(* IEC 61131-3 sources: Industry-PLC-LLM/data/PLCBEAD_repo/PLCBEAD_PLCEmbed-main/PLC-BEAD/Source/GEB/SWAP_BYTE, 1 file *)

(* ---- SWAP_BYTE.ST ---- *)
FUNCTION SWAP_BYTE:WORD

	VAR_INPUT
		IN :	WORD;
	END_VAR

	Swap_Byte := ROL(IN,8);

END_FUNCTION

PROGRAM program0

	VAR
		IN :	WORD;
		CEIL5_OUT : WORD;
	END_VAR

	CEIL5_OUT := SWAP_BYTE(IN);

END_PROGRAM
